Fanuc KAREL source: kb00171.KL

-- PROVISIONAL review KL for V770-1; original PC SHA256 a20e58d3c84067160e8977287f186b6a13ee80c0339d66a81d5d402ad1deb218
-- Incomplete behavior may be omitted. Consult companion uncertainty JSON. Do not deploy.
PROGRAM KB00171
%NOLOCKGROUP
BEGIN
  -- UNRESOLVED_PC offsets 5-12; opcodes 9D,23
  -- UNRESOLVED_PC offsets 17-24; opcodes 9D,23
  -- UNRESOLVED_PC offsets 29-36; opcodes 9D,23
  -- UNRESOLVED_PC offsets 41-69; opcodes 27,22,22,22,31,23
  -- UNRESOLVED_PC offsets 74-78; opcodes 7F
END KB00171
